{attribute 'pack_mode' := '2'}
TYPE ST_NCI_CTRL :
STRUCT
  eCmd          : E_NCI_CTRL := E_NCI_CTRL.INIT;
  rOverride     : REAL := 47.11;

  sProgramName  : STRING(255);
END_STRUCT
END_TYPE

(* stored: Version 1.1.0.1
   DUT ST_NCI_CTRL: Id {9175a094-7a51-4c4c-9afd-a383ff198f39} *)
